INTERFACE I_Header

METHOD PUBLIC ToString
VAR_INPUT
	Destination : REFERENCE TO STRING(ServerConfiguration.HEADER_STRING_SIZE);
END_VAR
END_METHOD

METHOD PUBLIC TryGetField : BOOL;
VAR_INPUT
	Key : STRING;
	Destination : ANY;
END_VAR
END_METHOD

METHOD PUBLIC TryWriteField : BOOL;
VAR_INPUT
	Key : STRING;
	Source : ANY;
END_VAR
END_METHOD

END_INTERFACE

(* stored: Version 1.1.0.1, ProductVersion 3.1.4026.13
   Itf I_Header: Id {932910ad-d278-49f7-a97d-c04d5f97460c}
   Method ToString: Id {c125b673-342a-4b80-8aa3-9d32af2f4197}
   Method TryGetField: Id {70478fd9-33e4-43c7-a3fd-eb4aad9b59d1}
   Method TryWriteField: Id {b20a2c1d-f5f9-4e2f-8a86-d676a15fad14} *)
